TYPE Signalbezeichnungen :
STRUCT
	Name: STRING;
END_STRUCT
END_TYPE

(* stored: Version 1.1.0.1, ProductVersion 3.1.4022.16
   DUT Signalbezeichnungen: Id {d7b3af49-48c2-44b9-abd0-60172f338b04} *)
